FUNCTION_BLOCK OneTestHasMissingTest EXTENDS FB_TestSuite

NameMatches();
MissingTestAtTheStart();

METHOD MissingTestAtTheStart
VAR_INPUT
END_VAR
AssertTrue(Condition:=TRUE, Message:='Blabla');

TEST_FINISHED();
END_METHOD

METHOD NameMatches
TEST('NameMatches');

AssertTrue(Condition:=TRUE, Message:='Blabla');

TEST_FINISHED();
END_METHOD

END_FUNCTION_BLOCK

(* stored: Version 1.1.0.1, ProductVersion 3.1.4024.12
   POU OneTestHasMissingTest: Id {bf8d71b6-a27f-4ba4-bb08-a3fc34e4409d}, SpecialFunc None
   Method MissingTestAtTheStart: Id {5e89dcb4-9304-45a7-8b6c-f944a99ca271}
   Method NameMatches: Id {1989bb87-271a-43c8-8920-4c9d0ddcf1e0} *)
